FUNCTION_BLOCK PUBLIC FB_DataBufferManager
VAR_INPUT
	ArraySize : INT;
	DataRepository : POINTER TO DataBuffer;	 // Element 0 for data preparation
END_VAR

METHOD Clear : BOOL
VAR_INPUT
	Position : INT := -1;
END_VAR
	IF (Position>0 AND Position<ArraySize) THEN
// Clear single position array repository  
		MEMSET(ADR(DataRepository[Position]), 16#00, SIZEOF(DataBuffer));
	ELSIF Position =-1 THEN
// Clear all position array	repository	
		MEMSET(ADR(DataRepository), 16#00, SIZEOF(DataRepository));
	ELSE
// Error
		;
	END_IF
END_METHOD

METHOD Ins : BOOL
VAR_INPUT
	DataIn: DataBuffer;
END_VAR
VAR
	i: UINT;
END_VAR
;
(*IF NOT DataRepository[0].PartState.Valid THEN
	MEMCPY(ADR(DataRepository[0]), ADR(DataIn), SIZEOF(DUT_PartData));	
ELSE
	// Error: GetNewPartData called with slot 0 non empty
END_IF*)

MEMCPY(ADR(DataRepository[0]), ADR(DataIn), SIZEOF(DataBuffer));
END_METHOD

METHOD M_Move : BOOL
VAR_INPUT
	DestPos		: UINT;
	SourcePos	: UINT;
END_VAR
IF DestPos >= 0 AND DestPos <= ArraySize AND SourcePos >=0 AND SourcePos <= ArraySize THEN
	MEMCPY(ADR(DataRepository[DestPos]), ADR(DataRepository[SourcePos]), SIZEOF(DataBuffer));
	
	MEMSET(ADR(DataRepository[SourcePos]), 16#00, SIZEOF(DataBuffer));
ELSE
	;//error
END_IF
END_METHOD

METHOD PUBLIC Read : BOOL
VAR_INPUT
	Position 	: UINT;
END_VAR

VAR_OUTPUT
	Dest		: DataBuffer;
END_VAR

//CASE Position OF
//	0..NUM_STAIONS:
//		MEMCPY(ADR(Dest), ADR(DataRepository[Position]), SIZEOF(DUT_PartData));
//ELSE	
//	;	// Error
//END_CASE

IF (Position>0 AND Position<20) THEN
		MEMCPY(ADR(Dest), ADR(DataRepository[Position]), SIZEOF(DataBuffer));
ELSE	
	;	// Error
END_IF
END_METHOD

METHOD PUBLIC Shift : BOOL
VAR
	i : UINT;
END_VAR
// Shift data array from StartPos(first data array moved) to EndPos (Last data array destination)
FOR i:= ArraySize TO 1 BY -1 DO
	MEMCPY(ADR(DataRepository[i]), ADR(DataRepository[i-1]), SIZEOF(DataBuffer));
END_FOR;

// Clear start position data array
MEMSET(ADR(DataRepository[0]), 16#00, SIZEOF(DataBuffer));
END_METHOD

METHOD PUBLIC ShiftRange : BOOL
VAR_INPUT
	StartPos	: INT;
	EndPos 		: INT;
END_VAR
VAR
	i : INT;
	N : INT := 0;
END_VAR
IF(StartPos < EndPos AND EndPos <= ArraySize) THEN
	N := EndPos - StartPos - 1;
	FOR i:= 0 TO N DO
		MEMCPY(ADR(DataRepository[EndPos-i]), ADR(DataRepository[EndPos-i-1]), SIZEOF(DataBuffer));
	END_FOR;
ELSE
	; //Error;
END_IF;

// Clear start position data array
MEMSET(ADR(DataRepository[StartPos]), 16#00, SIZEOF(DataBuffer));
END_METHOD

METHOD Update : BOOL
VAR_INPUT
END_VAR
// TODO: GraphQL mutation with FIFO
END_METHOD

END_FUNCTION_BLOCK

(* stored: Version 1.1.0.1, ProductVersion 3.1.4024.15
   POU FB_DataBufferManager: Id {e35cddbb-778f-4c3a-a571-ed8d99eb504e}, SpecialFunc None
   Method Clear: Id {1b54d676-330e-4a9c-b7fe-4a1e6618443c}
   Method Ins: Id {6e9e10cd-b241-44cb-a616-1081af818a04}
   Method M_Move: Id {9cd92544-2d8f-4db2-8c0c-777b5aa8aea3}
   Method Read: Id {df885a84-945e-46fe-a85c-b11aa4c0ebd5}
   Method Shift: Id {34128583-968f-41ec-8113-305f13bb64ca}
   Method ShiftRange: Id {e67c0dc7-0613-4b98-9903-fc791aae9f40}
   Method Update: Id {20205ed3-1e1a-4e7a-b271-7508b35f0ef9} *)
